// TIA Portal V14 SP1 export
// export: Created 2019-05-09T00:36:17.8690758Z, ExportSetting None, DisplayName Totally Integrated Automation Portal, DisplayVersion V14 SP1 Update 7, DisplayName TIA Portal Openness, DisplayVersion V14 SP1 Update 6, DisplayName STEP 7 Basic, DisplayVersion V14 SP1 Update 7, DisplayName WinCC Basic, DisplayVersion V14 SP1 Update 7
ORGANIZATION_BLOCK "Main"   // OB1, LAD, ProgramCycle
TITLE = "Main Program Sweep (Cycle)"
{ S7_Optimized_Access := 'TRUE' }
   VAR_INPUT
      Initial_Call : Bool;   // Initial call of this OB
      Remanence : Bool;   // =True, if remanent data are available
   END_VAR
BEGIN

REGION Network 1
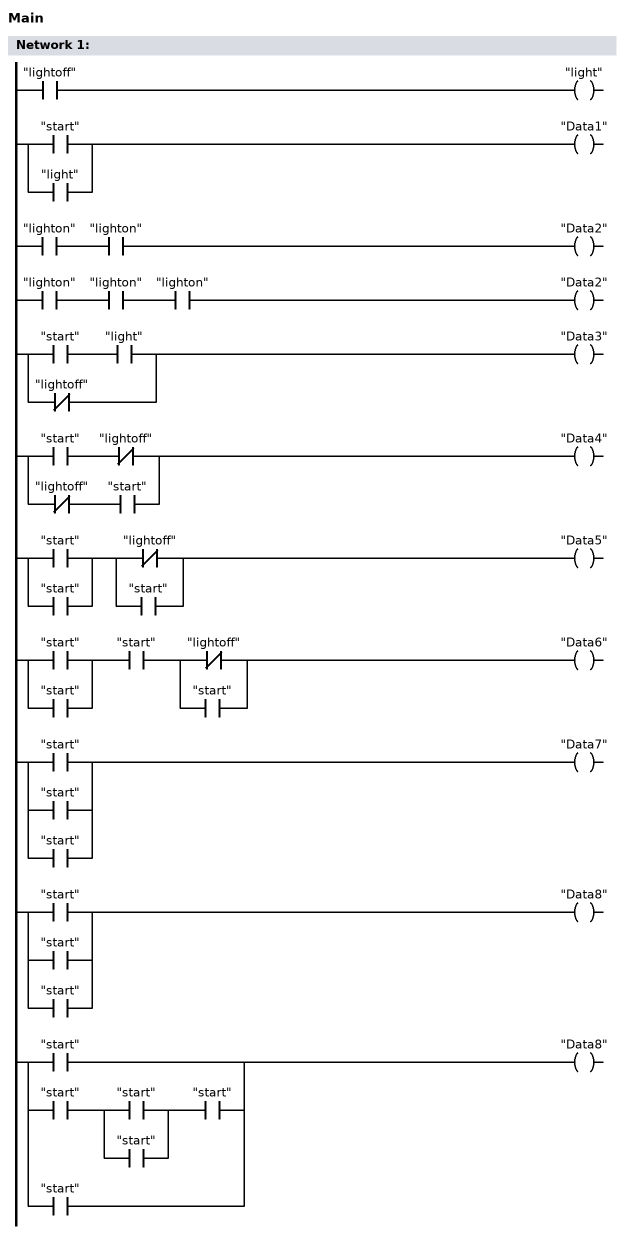
   RUNG wire#powerrail
      Contact( "lightoff" )
      Coil( "light" )
   END_RUNG
   RUNG wire#powerrail
      Contact( "start" )
      wire#w1
      Coil( "Data1" )
   END_RUNG
   RUNG wire#powerrail
      Contact( "light" )
   END_RUNG wire#w1
   RUNG wire#powerrail
      Contact( "lighton" )
      Contact( "lighton" )
      Coil( "Data2" )
   END_RUNG
   RUNG wire#powerrail
      Contact( "lighton" )
      Contact( "lighton" )
      Contact( "lighton" )
      Coil( "Data2" )
   END_RUNG
   RUNG wire#powerrail
      Contact( "start" )
      Contact( "light" )
      wire#w2
      Coil( "Data3" )
   END_RUNG
   RUNG wire#powerrail
      I_Contact( "lightoff" )
   END_RUNG wire#w2
   RUNG wire#powerrail
      Contact( "start" )
      I_Contact( "lightoff" )
      wire#w3
      Coil( "Data4" )
   END_RUNG
   RUNG wire#powerrail
      I_Contact( "lightoff" )
      Contact( "start" )
   END_RUNG wire#w3
   RUNG wire#powerrail
      Contact( "start" )
      wire#w4
      I_Contact( "lightoff" )
      wire#w5
      Coil( "Data5" )
   END_RUNG
   RUNG wire#powerrail
      Contact( "start" )
   END_RUNG wire#w4
   RUNG wire#w4
      Contact( "start" )
   END_RUNG wire#w5
   RUNG wire#powerrail
      Contact( "start" )
      wire#w6
      Contact( "start" )
      wire#w7
      I_Contact( "lightoff" )
      wire#w8
      Coil( "Data6" )
   END_RUNG
   RUNG wire#powerrail
      Contact( "start" )
   END_RUNG wire#w6
   RUNG wire#w7
      Contact( "start" )
   END_RUNG wire#w8
   RUNG wire#powerrail
      Contact( "start" )
      wire#w9
      Coil( "Data7" )
   END_RUNG
   RUNG wire#powerrail
      Contact( "start" )
   END_RUNG wire#w9
   RUNG wire#powerrail
      Contact( "start" )
   END_RUNG wire#w9
   RUNG wire#powerrail
      Contact( "start" )
      wire#w10
      Coil( "Data8" )
   END_RUNG
   RUNG wire#powerrail
      Contact( "start" )
   END_RUNG wire#w10
   RUNG wire#powerrail
      Contact( "start" )
   END_RUNG wire#w10
   RUNG wire#powerrail
      Contact( "start" )
      wire#w11
      Coil( "Data8" )
   END_RUNG
   RUNG wire#powerrail
      Contact( "start" )
      wire#w12
      Contact( "start" )
      wire#w13
      Contact( "start" )
   END_RUNG wire#w11
   RUNG wire#w12
      Contact( "start" )
   END_RUNG wire#w13
   RUNG wire#powerrail
      Contact( "start" )
   END_RUNG wire#w11
   // the same network as SCL:
   "light" := "lightoff";
   "Data1" := "start" OR "light";
   "Data2" := "lighton" AND "lighton";
   "Data2" := "lighton" AND "lighton" AND "lighton";
   "Data3" := ("start" AND "light") OR NOT "lightoff";
   "Data4" := ("start" AND NOT "lightoff") OR (NOT "lightoff" AND "start");
   "Data5" := ("start" OR "start") AND (NOT "lightoff" OR "start");
   "Data6" := ("start" OR "start") AND "start" AND (NOT "lightoff" OR "start");
   "Data7" := "start" OR "start" OR "start";
   "Data8" := "start" OR "start" OR "start";
   "Data8" := "start" OR ("start" AND ("start" OR "start") AND "start") OR "start";
END_REGION
END_ORGANIZATION_BLOCK
